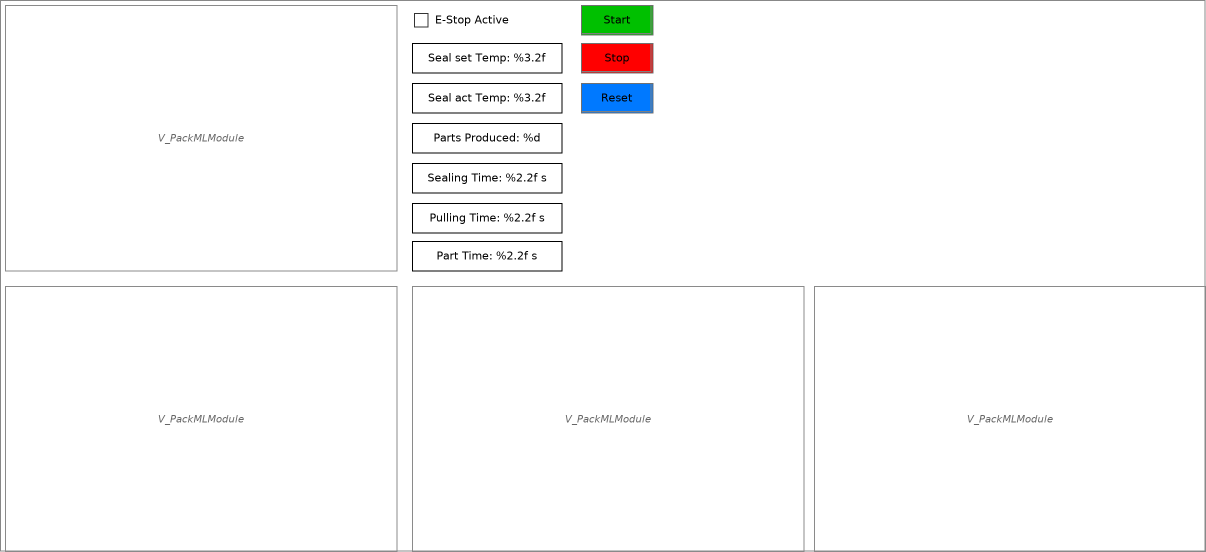
VISUALIZATION V_Main  // 1206x552
    Checkbox (412,5 150x30), "E-Stop Active", variable: MAIN.VFFS.EStop1_Pressed
    Frame (5,5 392x266)
        shows V_PackMLModule(PackML_HMI := MAIN.VFFS.VFFS_HMI.Statemachine_HMI)
    Frame (5,286 392x266)
        shows V_PackMLModule(PackML_HMI := MAIN.VFFS._PullWheels.Statemachine_HMI.Statemachine_HMI)
    Frame (412,286 392x266)
        shows V_PackMLModule(PackML_HMI := MAIN.VFFS._Sealer.Statemachine_HMI.Statemachine_HMI)
    Frame (814,286 392x266)
        shows V_PackMLModule(PackML_HMI := MAIN.VFFS._Unwind.Statemachine_HMI.Statemachine_HMI)
    Rectangle (412,43 150x30), "Seal set Temp: %3.2f", text variable: MAIN.VFFS._Sealer._SealBar._SetTemperature
    Rectangle (412,83 150x30), "Seal act Temp: %3.2f", text variable: MAIN.VFFS._Sealer._SealBar._ActualTemperature
    Rectangle (412,123 150x30), "Parts Produced: %d", text variable: MAIN.VFFS._PartsProduced
    Button (581,5 72x30), "Start", input disabled if: NOT MAIN.VFFS.VFFS_HMI.Statemachine_HMI.StartPermissive
        OnMouseDown: execute { MAIN.VFFS.VFFS_HMI.Statemachine_HMI.StartPressed := TRUE; }
        OnMouseUp: execute { MAIN.VFFS.VFFS_HMI.Statemachine_HMI.StartPressed := FALSE; }
    Button (581,43 72x30), "Stop", input disabled if: NOT MAIN.VFFS.VFFS_HMI.Statemachine_HMI.StopPermissive
        OnMouseDown: execute { MAIN.VFFS.VFFS_HMI.Statemachine_HMI.StopPressed := TRUE; }
        OnMouseUp: execute { MAIN.VFFS.VFFS_HMI.Statemachine_HMI.StopPressed := False; }
    Button (581,83 72x30), "Reset", input disabled if: NOT MAIN.VFFS.VFFS_HMI.Statemachine_HMI.ResetPermissive
        OnMouseDown: execute { MAIN.VFFS.VFFS_HMI.Statemachine_HMI.ResetPressed := TRUE; }
        OnMouseUp: execute { MAIN.VFFS.VFFS_HMI.Statemachine_HMI.ResetPressed := FALSE; }
    Rectangle (412,163 150x30), "Sealing Time: %2.2f s", text variable: MAIN.VFFS._SealingTime
    Rectangle (412,203 150x30), "Pulling Time: %2.2f s", text variable: MAIN.VFFS._PullingTime
    Rectangle (412,241 150x30), "Part Time: %2.2f s", text variable: MAIN.VFFS._PartTime
END_VISUALIZATION

(* stored: Version 1.1.0.1, ProductVersion 3.1.4026.18
   Visu V_Main: Id {fe59b201-0f2d-4510-87ae-935987371194} *)
